VAR_GLOBAL
    bMasterReset: BOOL;                               // Sistem master reset
END_VAR

(* stored: Version 1.1.0.1, ProductVersion 3.1.4024.15
   GVL GVL_System: Id {b0bebe06-de5b-4958-9d15-5240a47dc133} *)
